FUNCTION NullLogger : I_Logger		// Returns a null logger instance

NullLogger := LOGGER.nullLogger;

END_FUNCTION

(* stored: Version 1.1.0.1, ProductVersion 3.1.4026.18
   POU NullLogger: Id {d92f1651-c559-4d36-bdc4-359e3585c04d}, SpecialFunc None *)
